{attribute 'qualified_only'}
VAR_GLOBAL
    // M1K3
    // Motors
    {attribute 'TcLinkTo' := '.bLimitForwardEnable:=TIIB[EL7047_M1K3_Yup]^STM Status^Status^Digital input 1;
                              .bLimitBackwardEnable:=TIIB[EL7047_M1K3_Yup]^STM Status^Status^Digital input 2'}
    {attribute 'pytmc' := '
        pv: MR1K3:SOMS:MMS:YUP
    '}
    M1 : DUT_MotionStage := (fVelocity:=100.0, nEnableMode:=ENUM_StageEnableMode.ALWAYS); // M1K3 Yup


    {attribute 'TcLinkTo' := '.bLimitForwardEnable:=TIIB[EL7047_M1K3_Ydwn]^STM Status^Status^Digital input 1;
                              .bLimitBackwardEnable:=TIIB[EL7047_M1K3_Ydwn]^STM Status^Status^Digital input 2'}
    {attribute 'pytmc' := '
        pv: MR1K3:SOMS:MMS:YDWN
    '}
    M2 : DUT_MotionStage := (fVelocity:=100.0, nEnableMode:=ENUM_StageEnableMode.ALWAYS); // M1K3 Ydwn


    {attribute 'TcLinkTo' := '.bLimitForwardEnable:=TIIB[EL7047_M1K3_Xup]^STM Status^Status^Digital input 1;
                              .bLimitBackwardEnable:=TIIB[EL7047_M1K3_Xup]^STM Status^Status^Digital input 2'}
    {attribute 'pytmc' := '
        pv: MR1K3:SOMS:MMS:XUP
    '}
    M3 : DUT_MotionStage := (fVelocity:=300.0, nEnableMode:=ENUM_StageEnableMode.ALWAYS); // M1K3 Xup


    {attribute 'TcLinkTo' := '.bLimitForwardEnable:=TIIB[EL7047_M1K3_Xdwn]^STM Status^Status^Digital input 1;
                              .bLimitBackwardEnable:=TIIB[EL7047_M1K3_Xdwn]^STM Status^Status^Digital input 2'}
    {attribute 'pytmc' := '
        pv: MR1K3:SOMS:MMS:XDWN
    '}
    M4 : DUT_MotionStage := (fVelocity:=300.0, nEnableMode:=ENUM_StageEnableMode.ALWAYS); // M1K3 Xdwn


    {attribute 'TcLinkTo' := '.bLimitForwardEnable:=TIIB[EL7047_M1K3_PitchCoarse]^STM Status^Status^Digital input 1;
                              .bLimitBackwardEnable:=TIIB[EL7047_M1K3_PitchCoarse]^STM Status^Status^Digital input 2'}
    {attribute 'pytmc' := '
        pv: MR1K3:SOMS:MMS:PITCH
    '}
    M5 : DUT_MotionStage := (fVelocity:=50.0); // M1K3 Pitch Stepper

    // M2K3
    // Motors
    {attribute 'TcLinkTo' := '.bLimitForwardEnable:=TIIB[EL7047_M2K3_Yup]^STM Status^Status^Digital input 1;
                              .bLimitBackwardEnable:=TIIB[EL7047_M2K3_Yup]^STM Status^Status^Digital input 2'}
    {attribute 'pytmc' := '
        pv: MR2K3:SOMS:MMS:YUP
    '}
    M6 : DUT_MotionStage := (fVelocity:=100.0, nEnableMode:=ENUM_StageEnableMode.ALWAYS); // M2K3 Yup


    {attribute 'TcLinkTo' := '.bLimitForwardEnable:=TIIB[EL7047_M2K3_Ydwn]^STM Status^Status^Digital input 1;
                              .bLimitBackwardEnable:=TIIB[EL7047_M2K3_Ydwn]^STM Status^Status^Digital input 2'}
    {attribute 'pytmc' := '
        pv: MR2K3:SOMS:MMS:YDWN
    '}
    M7 : DUT_MotionStage := (fVelocity:=100.0, nEnableMode:=ENUM_StageEnableMode.ALWAYS); // M2K3 Ydwn


    {attribute 'TcLinkTo' := '.bLimitForwardEnable:=TIIB[EL7047_M2K3_Xup]^STM Status^Status^Digital input 1;
                              .bLimitBackwardEnable:=TIIB[EL7047_M2K3_Xup]^STM Status^Status^Digital input 2'}
    {attribute 'pytmc' := '
        pv: MR2K3:SOMS:MMS:XUP
    '}
    M8 : DUT_MotionStage := (fVelocity:=150.0, nEnableMode:=ENUM_StageEnableMode.ALWAYS); // M2K3 Xup


    {attribute 'TcLinkTo' := '.bLimitForwardEnable:=TIIB[EL7047_M2K3_Xdwn]^STM Status^Status^Digital input 1;
                              .bLimitBackwardEnable:=TIIB[EL7047_M2K3_Xdwn]^STM Status^Status^Digital input 2'}
    {attribute 'pytmc' := '
        pv: MR2K3:SOMS:MMS:XDWN
    '}
    M9 : DUT_MotionStage := (fVelocity:=150.0, nEnableMode:=ENUM_StageEnableMode.ALWAYS); // M2K3 Xdwn


    {attribute 'TcLinkTo' := '.bLimitForwardEnable:=TIIB[EL7047_M2K3_PitchCoarse]^STM Status^Status^Digital input 1;
                              .bLimitBackwardEnable:=TIIB[EL7047_M2K3_PitchCoarse]^STM Status^Status^Digital input 2'}
    {attribute 'pytmc' := '
        pv: MR2K3:SOMS:MMS:PITCH
    '}
    M10 : DUT_MotionStage := (fVelocity:=50.0, nEnableMode:=ENUM_StageEnableMode.ALWAYS); // M2K3 Pitch Stepper

END_VAR

(* stored: Version 1.1.0.1, ProductVersion 3.1.4024.12
   GVL Main: Id {412255a3-a553-48c6-90ce-ed4007369e5b} *)
